(* PLC project Programme MGS_2-07_refactorJOY.project, CODESYS CODESYS V3.5 SP19 Patch 1 *)
(* stored: creationDateTime 2026-06-29T23:37:41.1378959, modificationDateTime 2026-06-29T22:49:33.424 *)

PROGRAM PRG_COD1
  VAR
    instFB_Encoder_Abs_0 : FB_Encoder_Abs;
    ratio : REAL;
  END_VAR

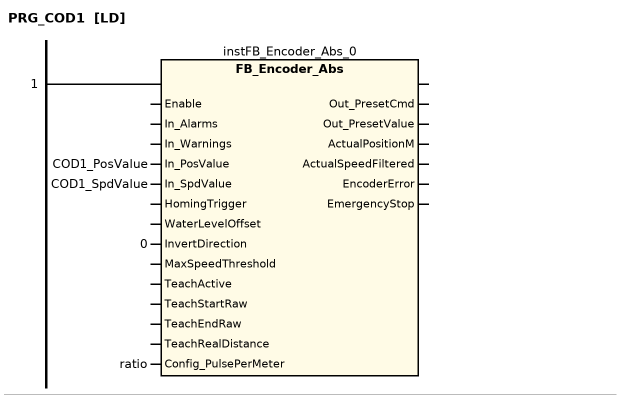
(* LD diagram, written out as Structured Text *)

instFB_Encoder_Abs_0(Enable := , In_Alarms := , In_Warnings := , In_PosValue := COD1_PosValue, In_SpdValue := COD1_SpdValue, HomingTrigger := , WaterLevelOffset := , InvertDirection := 0, MaxSpeedThreshold := , TeachActive := , TeachStartRaw := , TeachEndRaw := , TeachRealDistance := , Config_PulsePerMeter := ratio);
END_PROGRAM
